{attribute 'qualified_only'}
VAR_GLOBAL
	
	px: MotorProxy;
	motors: ARRAY[0..3] OF Motor;
END_VAR

(* stored: Version 1.1.0.1, ProductVersion 3.1.4024.13
   GVL GVL: Id {1be0b2ad-4ec8-47e1-b313-106b49c85b10} *)
